{attribute 'qualified_only'}
{attribute 'strict'}
TYPE E_PrimeSolventState :
(
	PS_Idle := 0,
    PS_Solvent1 := 10,
    PS_Solvent2 := 20,
    PS_Solvent3 := 30,
    PS_Solvent4 := 40,
    PS_Completed := 100
);
END_TYPE

(* stored: Version 1.1.0.1, ProductVersion 3.1.4024.15
   DUT E_PrimeSolventState: Id {38fe8732-9805-480d-8162-9790170dbcf9} *)
